FUNCTION_BLOCK TmsEmbarkStation EXTENDS Station IMPLEMENTS ITF_SwitchStation
VAR
	DepartMover : I_XtsMover;
	Axis : AXIS_REF;
	SwitchAxis : Axis_Base(Axis);
	_switchUpperPosition : MC_LREAL;
	_switchLowerPosition : MC_LREAL;
	ExecuteSequence : BOOL;
	_TrackLevel : INT := 1; //1 is low, 2 is high
	State :(
		Init,                                               
		Ready,                                 
        Waiting,
		HasSwitch,
		Call,
		FindTarget,
		Boarding,
		BoardingComplete,
		ActivateTrackForMover,
		Moving,
		Done,
		Aborting); 
	_switchPosition: MC_LREAL;
	arrTrackIds : ARRAY[1..2] OF I_XtsTrack;
	isUpAllowed : BOOL := TRUE;
	isDownAllowed : BOOL := FALSE;
	isMiddleAllowed : BOOL := TRUE;
	_BoardVelocity : MC_LREAL;
	_SwitchVelocity : MC_LREAL;
END_VAR

{analysis -2}

PROPERTY BoardVelocity : MC_LREAL
GET
BoardVelocity := _BoardVelocity;
END_GET
SET
_BoardVelocity := BoardVelocity;
END_SET
END_PROPERTY

METHOD PUBLIC  Cycle : HRESULT
VAR
	ActivateTrackResult : BOOL;
	BoardMoverResult : HRESULT;
	BaseCallResult : HRESULT;
END_VAR
Cycle := S_OK;
CASE State OF
	Init:
		_Operating := _Empty := _Complete := _Ready := _HasMover := FALSE;
		StationMovers := 0;
		State := Ready;
	
	Ready:	
		IF ExecuteSequence THEN
			_Operating := _Complete := _HasMover := FALSE;
			_Empty := _Ready := TRUE;
			StationMovers := 0;
			State := Waiting;
		END_IF
	
	Waiting:
		IF _HasMover THEN
			State := HasSwitch;
			_Operating := TRUE;
			_Empty := FALSE;
			_Ready := FALSE;
			_Complete := FALSE;
		END_IF
	
	HasSwitch:
		IF (_TrackLevel = 1 AND (SwitchAxis.isAtPosition(_switchLowerPosition) ))
			OR (_TrackLevel = 2 AND (SwitchAxis.isAtPosition(_switchUpperPosition))) THEN
					State := Boarding;
		ELSE
			State := Call;
		END_IF	
		
	Call:
		IF SwitchAxis.IsStationary() THEN
			IF _TrackLevel = 1 THEN
				SwitchAxis.MoveToPosition(Position := _switchLowerPosition, Velocity := _SwitchVelocity);
			ELSE
				SwitchAxis.MoveToPosition(Position := _switchUpperPosition, Velocity := _SwitchVelocity);
			END_IF
		ELSE
			State := Waiting;
		END_IF
			
	Boarding:
		BoardMoverResult := DepartMover.MoveTo(RequiredPosition := _switchPosition, MoveVelocity := _BoardVelocity, NonModuloMove := TRUE);
		IF DepartMover.isMoverAtPosition(position := _switchPosition) THEN
			State := BoardingComplete;
		END_IF
		
	BoardingComplete:
		IF _TrackLevel = 1 THEN
			SwitchAxis.MoveToPosition(Position := _switchUpperPosition, Velocity := _SwitchVelocity);
		ELSE
			SwitchAxis.MoveToPosition(Position := _switchLowerPosition, Velocity := _SwitchVelocity);
		END_IF
		State := BoardingComplete;
		
	Moving:
		IF (_TrackLevel = 1 AND SwitchAxis.isAtPosition(position := _switchUpperPosition)) OR
			(_TrackLevel = 2 AND SwitchAxis.isAtPosition(position := _switchLowerPosition)) THEN
			State := ActivateTrackForMover;
		END_IF
		
	ActivateTrackForMover:
		IF _TrackLevel = 1 THEN
			DepartMover.ActivateTrack(NewTrack := arrTrackIds[2].MyOTCID, Track := arrTrackIds[2]);
		ELSE
			DepartMover.ActivateTrack(NewTrack := arrTrackIds[1].MyOTCID, Track := arrTrackIds[1]);
		END_IF
		State := Moving;
		_Complete := TRUE;
			
	Done:
		IF _Complete AND NOT _HasMover THEN
			_Operating := FALSE;
			_Empty := TRUE;
			_Ready := TRUE;
			State := Waiting;
		END_IF	

	Aborting:
		State := Ready;	
		DepartMover := 0;
	ELSE
		Cycle := E_FAIL;
END_CASE
BaseCallResult := SUPER^.Cycle();
SwitchAxis.Cycle();
END_METHOD

METHOD HasMover : BOOL
VAR_INPUT
	mover : I_XtsMover;
END_VAR
IF StationMovers <= 2 THEN
	StationMovers := StationMovers + 1;
	DepartMover := mover;
	_HasMover := TRUE;
END_IF
HasMover := TRUE;
END_METHOD

METHOD PUBLIC MoverAway : BOOL
VAR_INPUT
END_VAR
StationMovers := StationMovers - 1;
IF StationMovers = 0 THEN
	_HasMover := FALSE;
END_IF
DepartMover := 0;
MoverAway := TRUE;
END_METHOD

METHOD StartSwitch : BOOL
VAR_INPUT
END_VAR
ExecuteSequence := TRUE;
END_METHOD

METHOD StopSwitch : BOOL
VAR_INPUT
END_VAR
ExecuteSequence := FALSE;
State := Aborting;
END_METHOD

PROPERTY SwitchLowerPosition : MC_LREAL
GET
END_GET
SET
END_SET
END_PROPERTY

METHOD PUBLIC SwitchMoveComplete : BOOL
VAR_INPUT
END_VAR
_Complete := TRUE;
SwitchMoveComplete := true;
END_METHOD

PROPERTY SwitchTravelPosition : mc_lreal
GET
SwitchTravelPosition := _switchPosition;
END_GET
SET
_switchPosition := SwitchTravelPosition;
END_SET
END_PROPERTY

PROPERTY SwitchUpperPosition : MC_LREAL
GET
END_GET
SET
END_SET
END_PROPERTY

PROPERTY TrackIds : array[1..2] of I_XtsTrack
GET
TrackIds := arrTrackIds;
END_GET
SET
arrTrackIds := TrackIds;
END_SET
END_PROPERTY

PROPERTY TrackLevel : INT
GET
TrackLevel := _TrackLevel;
END_GET
SET
_TrackLevel := TrackLevel;
END_SET
END_PROPERTY

END_FUNCTION_BLOCK

(* stored: Version 1.1.0.1
   POU TmsEmbarkStation: Id {4d15a973-29cb-4ffe-934a-8f072d992ec0}, SpecialFunc None
   Property BoardVelocity: Id {af5577ef-90f6-4070-9e3d-dce62d068c94}
   Get Get: Id {442f20d9-4d5c-462e-ace0-37721614361e}
   Set Set: Id {4f476cb8-1c36-46ee-b33f-8098bec190be}
   Method Cycle: Id {30dc7518-cfa1-45c8-85d7-d03d0ef4ae28}
   Method HasMover: Id {466b4750-cbf0-42df-80f2-b3d4852756ba}
   Method MoverAway: Id {45498adf-6827-4a97-8c80-ff53aebb1724}
   Method StartSwitch: Id {c29e9395-8979-4e9a-90a8-1d97909d0ac9}
   Method StopSwitch: Id {3cacf78b-01e4-4c36-b301-1826803c65db}
   Property SwitchLowerPosition: Id {190ee51d-8616-4771-bea0-4a043a7d3d59}
   Get Get: Id {2179123a-03ea-4eb3-8d32-50c09c60e6da}
   Set Set: Id {98459ca6-5c5e-4646-8d93-b28fde23c27f}
   Method SwitchMoveComplete: Id {a8eedfd9-7707-47a4-b55d-1e335fa7f41f}
   Property SwitchTravelPosition: Id {506615ae-e584-4b6b-8c90-23702c945ca0}
   Get Get: Id {770e482e-e926-4e26-8349-fb06dc2d74be}
   Set Set: Id {2f71d79c-8b57-4fda-9b2a-e631ae1faffd}
   Property SwitchUpperPosition: Id {5e471955-b1fa-42e8-8457-954969d80adc}
   Get Get: Id {6218b073-eaf9-44e9-8692-abdac10dd02b}
   Set Set: Id {5e38ec9d-d9b7-4541-b1f9-c48e79167e2a}
   Property TrackIds: Id {061f1ace-88f0-4461-91e3-203af1d3961d}
   Get Get: Id {eb5d1a17-a69b-486a-bd32-b1fce0797a7b}
   Set Set: Id {f6abe2e3-3d9c-4b6c-81bd-f3b0563c7882}
   Property TrackLevel: Id {3cbcc021-27ff-4251-b3d2-761cf34c192e}
   Get Get: Id {eac07d3d-cc95-4d94-be8d-aab0ced9fdea}
   Set Set: Id {4b1478e4-977e-454a-a0bf-fe888f795dfb} *)
